// TIA Portal V16 export
// export: Created 2021-04-11T09:51:29.8490423Z, ExportSetting WithDefaults, DisplayName Totally Integrated Automation Portal, DisplayVersion V16, DisplayName TIA Portal Version Control Interface, DisplayVersion V16, DisplayName TIA Portal Openness, DisplayVersion V16, DisplayName STEP 7 Professional, DisplayVersion V16, DisplayName STEP 7 Safety, DisplayVersion V16, DisplayName WinCC Unified SCADA Engineering System, DisplayVersion V16
TYPE "LineWeight"
// stored: IsFailsafeCompliant false
   STRUCT
      isVibroLotWork : Bool;   // работа вибролотка
      percentVibroLot : Int;   // текущая вибрация вибролотка
      stateValveAfterVibroLot : Bool;   // состояние закрылки после вибролотка
      stateLeftValveWeightPocket : Bool;   // состояние левого клапана открывающегося кармана
      stateRightValveWeightPocket : Bool;   // состояние правого клапана открывающегося кармана
      targetWeightPocket : Real;   // целевой вес кармана
      currentWeightPocket : Real;   // текущий вес в кармане
      manOpenValveAfterVibroLot : Bool;   // ручн - открыть лопатку
      manCloseValveAfterVibroLot : Bool;   // ручн - закрыть лопатку
      manOpenLeftValveWeightPocket : Bool;   // ручн -открыть левый карман
      manCloseLeftValveWeightPocket : Bool;   // ручн -закрыть левый карман
      manOpenRightValveWeightPocket : Bool;   // ручн - открыть правый карман
      manCloseRightValveWieghtPocket : Bool;   // ручн - закрыть правый карман
      manVibroLotStart : Bool;   // ручн - управление ПУСК\Стоп вибролотка
      begWeightModuleReady : Bool;   // начальный экран - готовность весоизмерительного модуля
   END_STRUCT;
END_TYPE
